//{attribute 'pack_mode' := '8'}
TYPE ST_HierarchyData :
STRUCT

	UnitQty 	: STRING(10);
	GTIN 		: T_CodeGTIN;
	EAN 		: STRING(20);
	BCODE9	: T_CodeBRAND;
END_STRUCT
END_TYPE

(* stored: Version 1.1.0.1
   DUT ST_HierarchyData: Id {f4fa1992-5070-43f0-a1cb-81cabd8dd48d} *)
